// LS Electric XG5000 project: 동남70
// PLC NewPLC
// module base 0 slot 0: 입출력 모듈:XBC-DN/DP14E (DC 24V 입력 8점, 트랜지스터 출력 6점)

PROGRAM NewProgram (task: 스캔 프로그램)

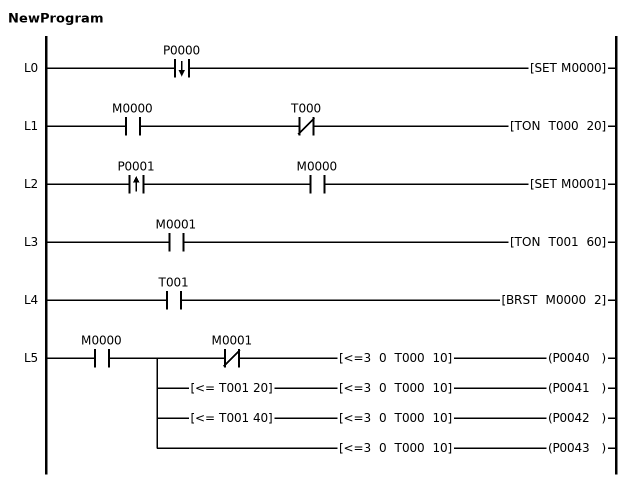
; L0
LOADN     P0000
SET       M0000
; L1
LOAD      M0000
AND NOT   T000
TON       T000 20
; L2
LOADP     P0001
AND       M0000
SET       M0001
; L3
LOAD      M0001
TON       T001 60
; L4
LOAD      T001
BRST      M0000 2
; L5
LOAD      M0000
MPUSH
AND NOT   M0001
AND<=3    0 T000 10
OUT       P0040
MLOAD
AND<=     T001 20
AND<=3    0 T000 10
OUT       P0041
MLOAD
AND<=     T001 40
AND<=3    0 T000 10
OUT       P0042
MPOP
AND<=3    0 T000 10
OUT       P0043